{attribute 'GeneratedUsingTerminal: KL2722'}
{attribute addProperty BoxType "KL2722"}
{attribute addProperty Description ""}
{attribute addProperty Physics ""}
{attribute addProperty Id "Channel_1AT %Q*Channel_460B8C400Channel_2AT %Q*Channel_460B8C400"}
{attribute addProperty CRC "3701954066"}
{attribute addProperty Size "0"}
TYPE KL2722_DCA75612 :
STRUCT
	{attribute addProperty Name "Channel_1"}
	Channel_1 : Channel_460B8C40;
	{attribute addProperty Name "Channel_2"}
	Channel_2 : Channel_460B8C40;
END_STRUCT
END_TYPE

(* stored: Version 1.2.0.0, ProductVersion 3.1.4024.9
   DUT KL2722_DCA75612: Id {e9a468f5-0ef0-4ba7-b413-207a75dc4a94} *)
